ABB RAPID module: CalibData.modx

MODULE CalibData
    ! PERS tooldata Servo:=[TRUE,[[0,0,114.2],[1,0,0,0]],[0.215,[8.7,12.3,49.2],[1,0,0,0],0.00021,0.00024,0.00009]];
    TASK PERS wobjdata Workobject_1:=[FALSE,TRUE,"",[[329.172,70.377,0],[1,0,0,0]],[[0,0,5],[1,0,0,0]]];
    TASK PERS wobjdata cube_storage :=[FALSE,TRUE,"",[[-705,35,950],[1,0,0,0]],[[0,0,5],[1,0,0,0]]];
   PERS tooldata Pen:=[TRUE,[[170.754,0.18,190.741],[0.653281482,-0.27059805,0.27059805,-0.653281482]],[0.25,[0,0,65],[1,0,0,0],0,0,0]];
    PERS tooldata Magnet:=[TRUE,[[-120.55,-0.18,140.537],[0.653281482,0.27059805,-0.27059805,-0.653281482]],[0.25,[0,0,65],[1,0,0,0],0,0,0]];
ENDMODULE
